(* Logix 5000 project; controller cal1615 1756-L62 rev 16.20; software revision 16.05; part 31 of 78 *)
(* tags used below, declared in another part *)
   AFI : BOOL;   // Always False Bit
   FAULT : BOOL;   // Fault AFI
   p01_param_fan_zero_speed : REAL;
   p01_param_open_oven_exh_sp : REAL;
   p01_param_open_oven_temp : REAL;
   p01_recipe_active : recipe;   // Active Recipe
   p01r09_open_oven : BOOL;
   p01r09_pb_global_reset : BOOL;   // System Modes PB: Global Fault Reset
   p02_dint_from_hmi : hmi_dint;
   p11r02_shutdown_temp : BOOL;   // Zone 1 Misc Control Safe Shutdown Temperature
   p11r30 : routine;   // Zone 1 Temperature Control
   p11r30_request_heat : BOOL;   // Zone 1 Temperature Control Request Heat
   p12r02_shutdown_temp : BOOL;   // Zone 2 Misc Control Safe Shutdown Temperature
   p12r30 : routine;   // Zone 2 Temperature Control
   p12r30_pid_temp : PID;   // Zone 2 Temperature Control PID
   p12r30_request_heat : BOOL;   // Zone 2 Temperature Control Request Heat
   p13_ai_exhaust_rpm : REAL;   // Zone 3 Analog Input Exhaust Fan RPM
   p13_ai_tc01 : REAL;   // Zone 3 Analog Input Control Thermocouple 1
   p13_ai_tc02 : REAL;   // Zone 3 Analog Input Control Thermocouple 2
   p13_ao_cv : REAL;   // Zone 3 Analog Output Control Valve
   p13_ao_exhaust_selected_speed : REAL;   // Zone 3 Analog Output Exhaust Fan VFD Selected Speed
   p13_di_door_open : BOOL;   // Zone 3 Digital Input Access Door Open
   p13_di_exh : acs800_di_normal;   // Zone 3 Digital Inputs Exhaust Fan
   p13_di_exh_fan_mtr_ts : BOOL;   // Zone 3 Digital Input Exhaust Fan Motor Thermostat OK
   p13_di_exh_flow_ok : BOOL;   // Zone 3 Digital Input Exhaust Flow OK
   p13_di_filter_clean : BOOL;   // Zone 3 Digital Input Filter Dirty
   p13_di_recirc : acs800_di_normal;   // Zone 3 Digital Inputs Recirc Fan
   p13_di_tc01_bo : BOOL;   // Zone 3 Digital Input Control Thermocouple 1 Failure
   p13_di_tc02_bo : BOOL;   // Zone 3 Digital Input Control Thermocouple 2 Failure
   p13_dint_to_hmi : DINT[16];   // Zone 3 Temperature Control VFDs On
   p13_do_exh : acs800_do_normal;   // Zone 3 Digital Output Exhaust Fan
   p13_param_pid2_ff : REAL;   // Zone 3 Parameter Auto PID Bias
   p13_param_pid2_kd : REAL;   // Zone 3 Parameter Auto PID Derivative Gain
   p13_param_pid2_ki : REAL;   // Zone 3 Parameter Auto PID Integral Gain
   p13_param_pid2_kp : REAL;   // Zone 3 Parameter Auto PID Proportional Gain
   p13_param_tc01_dev : REAL;   // Zone 3 Parameter Oven Temperature Deviation from Setpoint
   p13r01 : routine;   // Zone 3 Main
   p13r02_shutdown_temp : BOOL;   // Zone 3 Misc Control Safe Shutdown Temperature
   p13r16_pid_temp_cv : DINT;   // Zone 3 Temperature Control Control Valve
   p13r20_state : DINT;   // Zone 3 Temperature Control State
   p13r30 : routine;   // Zone 3 Temperature Control
   p13r30_cv_man_sp : REAL;   // Zone 3 Temperature Control Manual Heat Control Valve Setpoint
   p13r30_pb_auto : BOOL;   // Zone 3 Temperature Control PB: Zone Control Auto
   p13r30_pb_manual : BOOL;   // Zone 3 Temperature Control PB: Zone Control Manual
   p13r30_pb_zone_off : BOOL;   // Zone 3 Temperature Control PB: Stop Zone Heat Control
   p13r30_pb_zone_on : BOOL;   // Zone 3 Temperature Control PB: Start Zone Heat Control
   p13r30_permissive_run : BOOL;   // Zone 3 Temperature Control Run Permissive
   p13r30_pid_temp_pv : REAL;   // Zone 3 Temperature Control PID Process Value
   p13r30_pid_temp_sp : REAL;   // Zone 3 Temperature Control PID Temperature Control Setpoint
   p13r30_pid_temp_sp_error : REAL;   // Zone 3 Temperature Control Setpoint/Process Variable Error (ABS)
   p13r30_pid_temp_sp_last : REAL;   // Zone 3 Temperature Control Setpoint Last Scan
   p13r30_request_cool : BOOL;   // Zone 3 Temperature Control Request Cooling
   p13r30_request_deviation_warning : BOOL;   // Zone 3 Temperature Control Request Setpoint Deviation Warning
   p13r30_request_manual : BOOL;   // Zone 3 Temperature Control Request Manual Control
   p13r30_request_PID_shot : BOOL;
   p13r30_temp_deviation_setpoint : DINT;
   p13r30_temp_pid_ctrl : PID;   // Zone 3 Temperature Control PID
   p13r30_timer_fault : TIMER[16];   // Zone 3 Temperature Control Fault Delay
   p13r30_timer_warning : TIMER[12];   // Zone 3 Temperature Control Warning Delay
   p13r30_vfds_ready : BOOL;   // Zone 3 Temperature Control VFDs On
   p13r31 : routine;   // Zone 3 Exhaust VFD
   p13r31_pb_start : BOOL;   // Zone 3 Exhaust VFD PB: Start
   p13r31_pb_stop : BOOL;   // Zone 3 Exhaust VFD PB: Stop
   p13r31_request_auto_run : BOOL;   // Zone 3 Exhaust Fan Run Request
   p13r31_run_permissive : BOOL;   // Zone 3 Exhaust VFD Run Permissive
   p13r31_timer_fault : TIMER[5];   // Zone 3 Exhaust VFD Fault Timer
   p13r31_timer_warning : TIMER[5];   // Zone 3 Exhaust VFD Waringing Timer
   p13r31_vfd_stopped : BOOL;   // Zone 3 Exhaust VFD VFD Stopped
   p23r02 : routine;   // Impreg Misc Control
(* P13_Zone_3, continued *)

ROUTINE R30_Temperature_Control   (* ladder *)
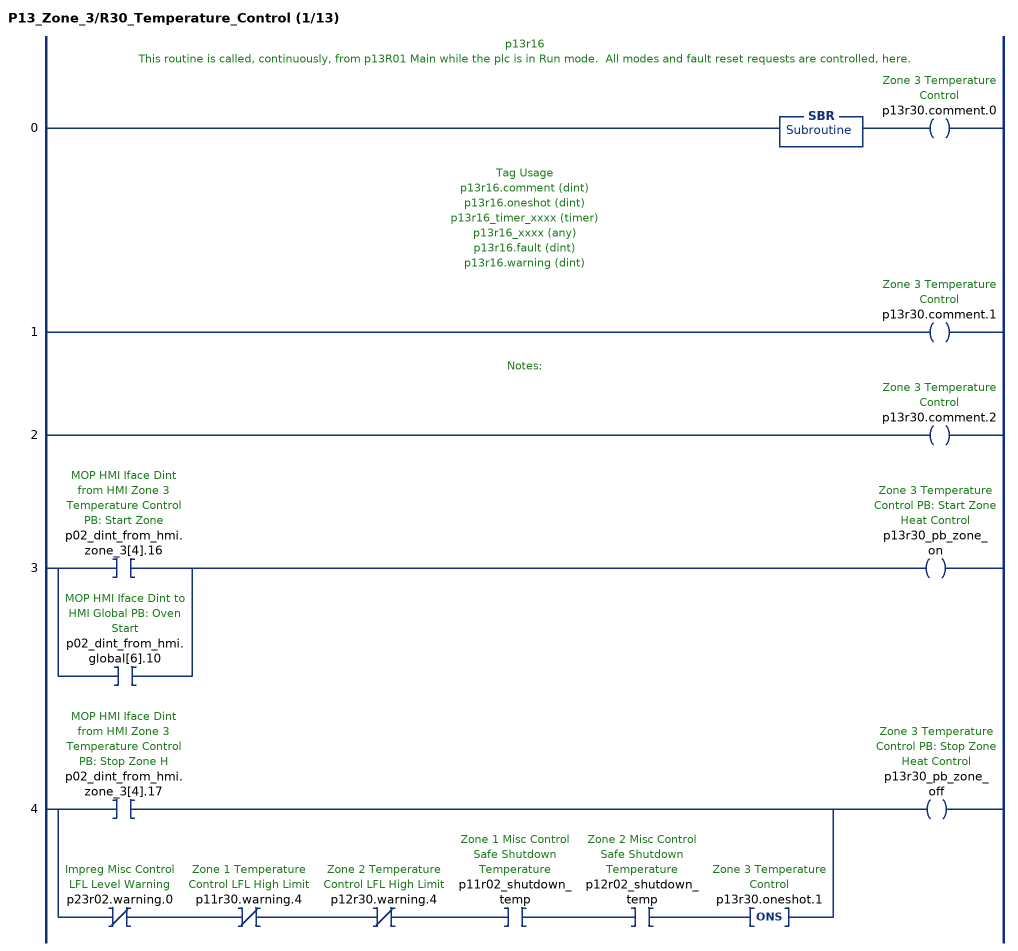
   // p13r16
   // This routine is called, continuously, from p13R01 Main while the plc is in Run mode.  All modes and fault reset requests are controlled, here.
   0: SBR()OTE(p13r30.comment.0);
   // Tag Usage
   // p13r16.comment (dint)
   // p13r16.oneshot (dint)
   // p13r16_timer_xxxx (timer)
   // p13r16_xxxx (any)
   // p13r16.fault (dint)
   // p13r16.warning (dint)
   1: OTE(p13r30.comment.1);
   // Notes:
   2: OTE(p13r30.comment.2);
   3: [XIC(p02_dint_from_hmi.zone_3[4].16) ,XIC(p02_dint_from_hmi.global[6].10) ]OTE(p13r30_pb_zone_on);
   4: [XIC(p02_dint_from_hmi.zone_3[4].17) ,XIO(p23r02.warning.0) XIO(p11r30.warning.4) XIO(p12r30.warning.4) XIC(p11r02_shutdown_temp) XIC(p12r02_shutdown_temp) ONS(p13r30.oneshot.1) ]OTE(p13r30_pb_zone_off);
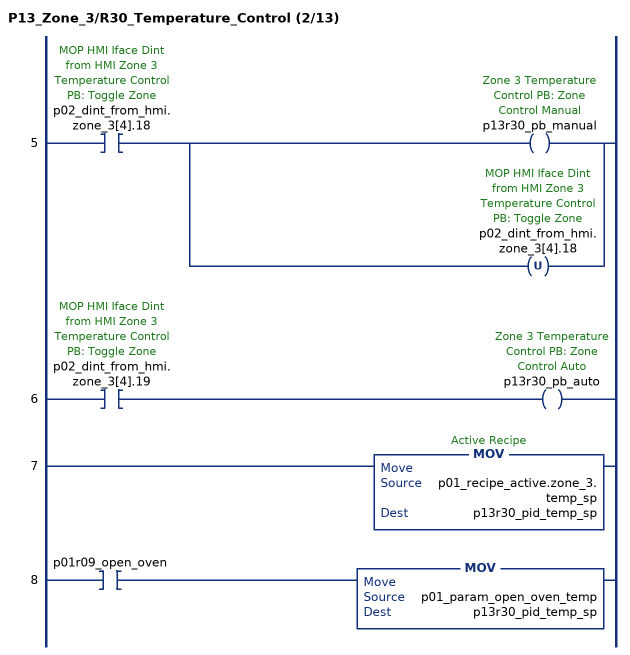
   5: XIC(p02_dint_from_hmi.zone_3[4].18)[OTE(p13r30_pb_manual) ,OTU(p02_dint_from_hmi.zone_3[4].18) ];
   6: XIC(p02_dint_from_hmi.zone_3[4].19)OTE(p13r30_pb_auto);
   7: MOV(p01_recipe_active.zone_3.temp_sp,p13r30_pid_temp_sp);
   8: XIC(p01r09_open_oven)MOV(p01_param_open_oven_temp,p13r30_pid_temp_sp);
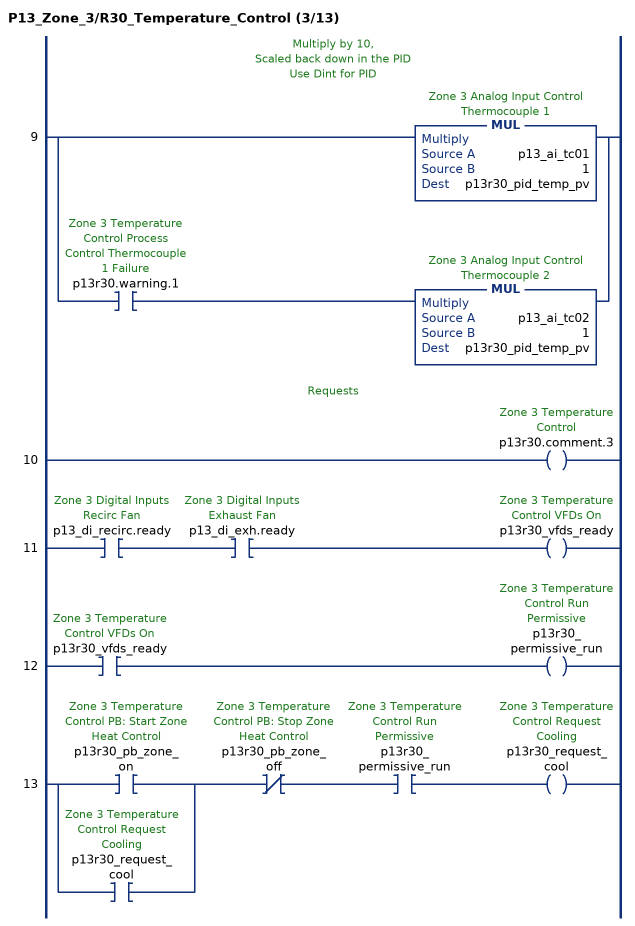
   // Multiply by 10,
   // Scaled back down in the PID
   // Use Dint for PID
   9: [MUL(p13_ai_tc01,1,p13r30_pid_temp_pv) ,XIC(p13r30.warning.1) MUL(p13_ai_tc02,1,p13r30_pid_temp_pv) ];
   // Requests
   10: OTE(p13r30.comment.3);
   11: XIC(p13_di_recirc.ready)XIC(p13_di_exh.ready)OTE(p13r30_vfds_ready);
   12: XIC(p13r30_vfds_ready)OTE(p13r30_permissive_run);
   13: [XIC(p13r30_pb_zone_on) ,XIC(p13r30_request_cool) ]XIO(p13r30_pb_zone_off)XIC(p13r30_permissive_run)OTE(p13r30_request_cool);
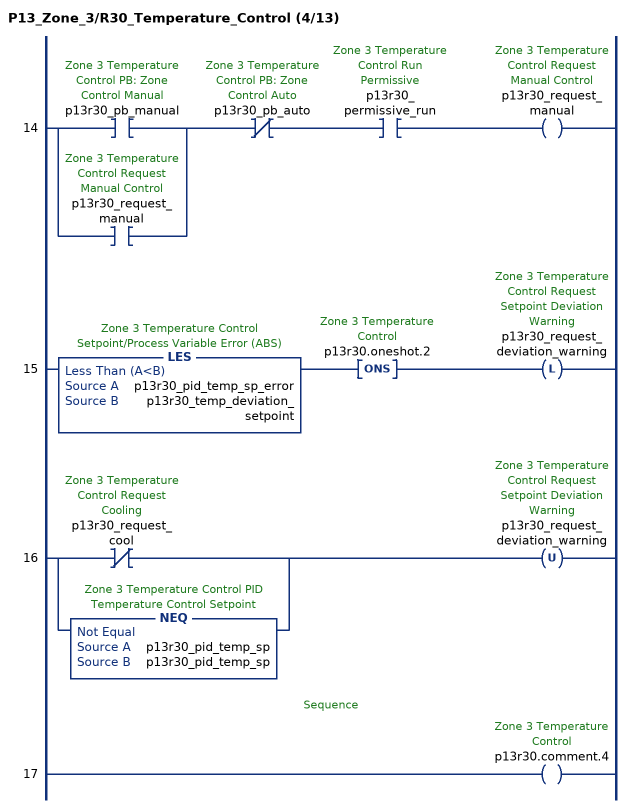
   14: [XIC(p13r30_pb_manual) ,XIC(p13r30_request_manual) ]XIO(p13r30_pb_auto)XIC(p13r30_permissive_run)OTE(p13r30_request_manual);
   15: LES(p13r30_pid_temp_sp_error,p13r30_temp_deviation_setpoint)ONS(p13r30.oneshot.2)OTL(p13r30_request_deviation_warning);
   16: [XIO(p13r30_request_cool) ,NEQ(p13r30_pid_temp_sp,p13r30_pid_temp_sp) ]OTU(p13r30_request_deviation_warning);
   // Sequence
   17: OTE(p13r30.comment.4);
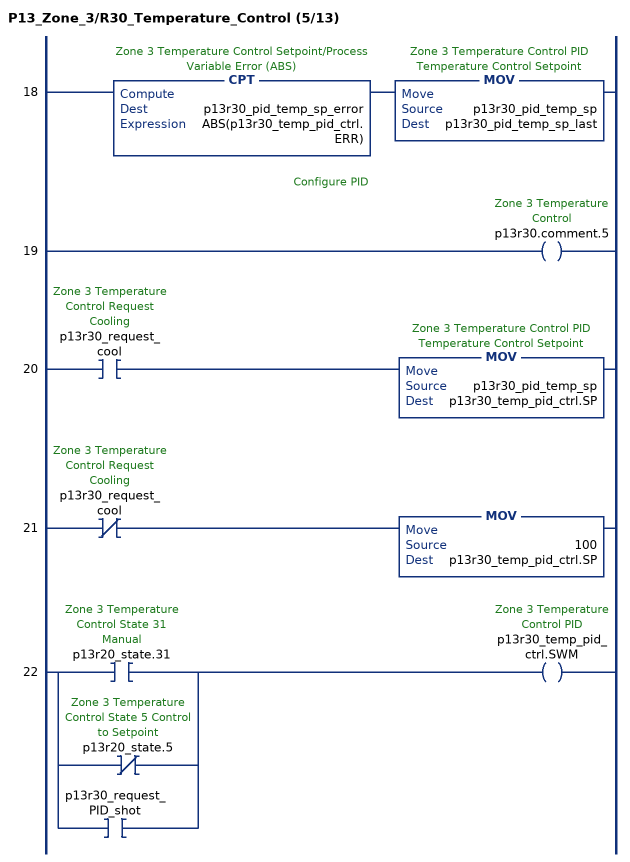
   18: CPT(p13r30_pid_temp_sp_error,ABS(p13r30_temp_pid_ctrl.ERR))MOV(p13r30_pid_temp_sp,p13r30_pid_temp_sp_last);
   // Configure PID
   19: OTE(p13r30.comment.5);
   20: XIC(p13r30_request_cool)MOV(p13r30_pid_temp_sp,p13r30_temp_pid_ctrl.SP);
   21: XIO(p13r30_request_cool)MOV(100,p13r30_temp_pid_ctrl.SP);
   22: [XIC(p13r20_state.31) ,XIO(p13r20_state.5) ,XIC(p13r30_request_PID_shot) ]OTE(p13r30_temp_pid_ctrl.SWM);
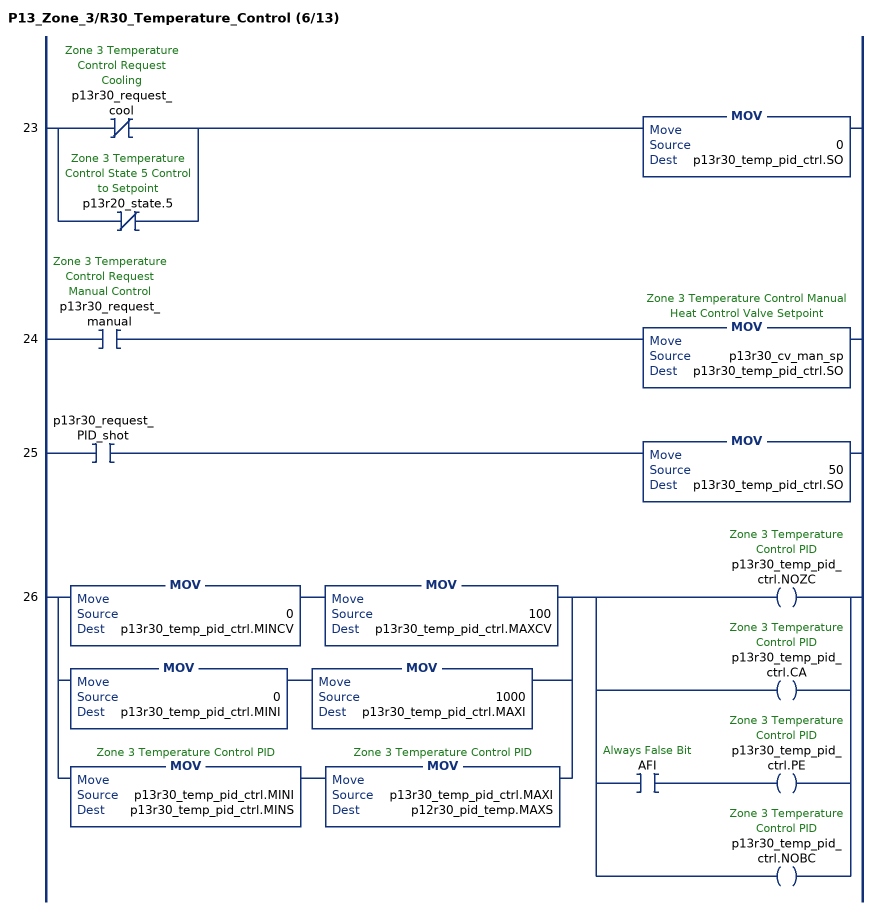
   23: [XIO(p13r30_request_cool) ,XIO(p13r20_state.5) ]MOV(0,p13r30_temp_pid_ctrl.SO);
   24: XIC(p13r30_request_manual)MOV(p13r30_cv_man_sp,p13r30_temp_pid_ctrl.SO);
   25: XIC(p13r30_request_PID_shot)MOV(50,p13r30_temp_pid_ctrl.SO);
   26: [MOV(0,p13r30_temp_pid_ctrl.MINCV) MOV(100,p13r30_temp_pid_ctrl.MAXCV) ,MOV(0,p13r30_temp_pid_ctrl.MINI) MOV(1000,p13r30_temp_pid_ctrl.MAXI) ,MOV(p13r30_temp_pid_ctrl.MINI,p13r30_temp_pid_ctrl.MINS) MOV(p13r30_temp_pid_ctrl.MAXI,p12r30_pid_temp.MAXS) ][OTE(p13r30_temp_pid_ctrl.NOZC) ,OTE(p13r30_temp_pid_ctrl.CA) ,XIC(AFI) OTE(p13r30_temp_pid_ctrl.PE) ,OTE(p13r30_temp_pid_ctrl.NOBC) ];
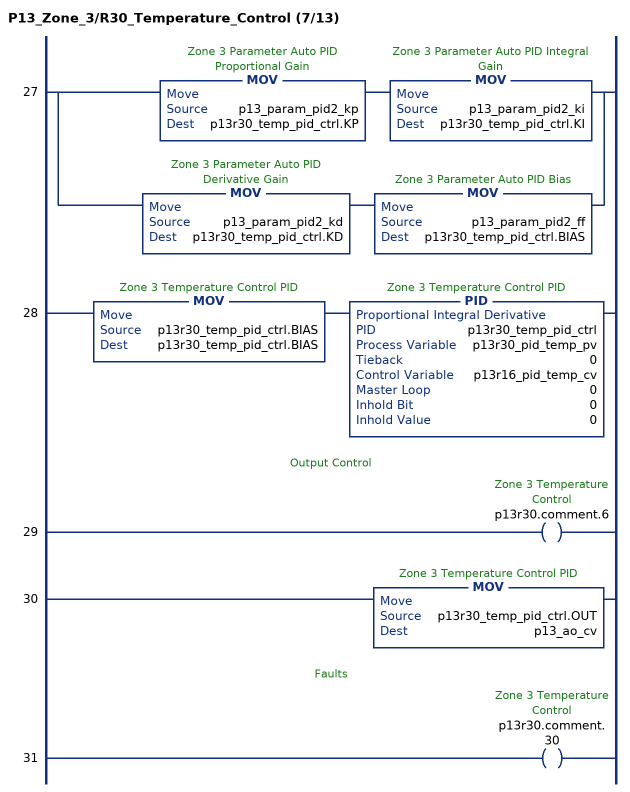
   27: [MOV(p13_param_pid2_kp,p13r30_temp_pid_ctrl.KP) MOV(p13_param_pid2_ki,p13r30_temp_pid_ctrl.KI) ,MOV(p13_param_pid2_kd,p13r30_temp_pid_ctrl.KD) MOV(p13_param_pid2_ff,p13r30_temp_pid_ctrl.BIAS) ];
   28: MOV(p13r30_temp_pid_ctrl.BIAS,p13r30_temp_pid_ctrl.BIAS)PID(p13r30_temp_pid_ctrl,p13r30_pid_temp_pv,0,p13r16_pid_temp_cv,0,0,0);
   // Output Control
   29: OTE(p13r30.comment.6);
   30: MOV(p13r30_temp_pid_ctrl.OUT,p13_ao_cv);
   // Faults
   31: OTE(p13r30.comment.30);
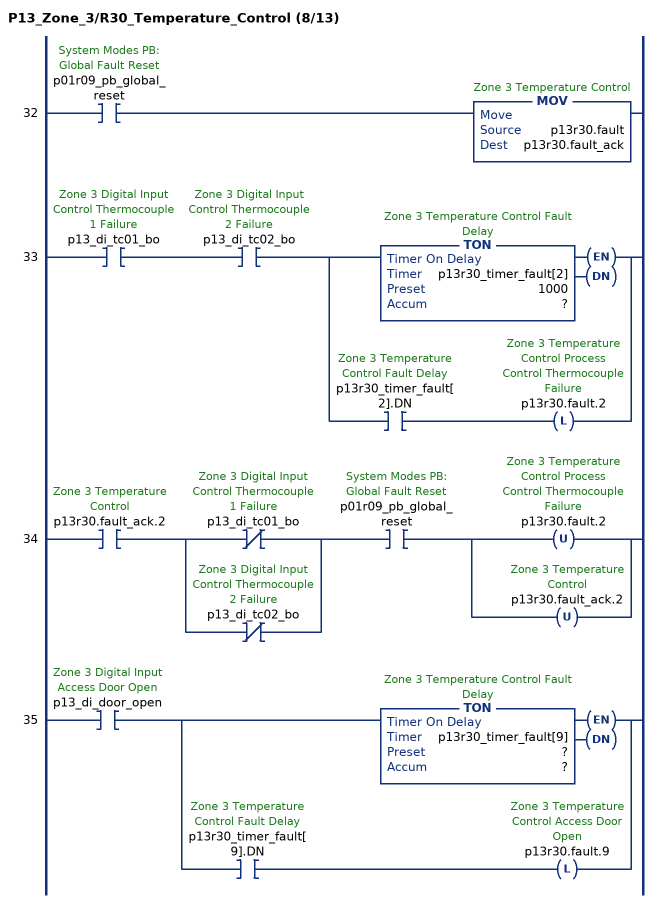
   32: XIC(p01r09_pb_global_reset)MOV(p13r30.fault,p13r30.fault_ack);
   33: XIC(p13_di_tc01_bo)XIC(p13_di_tc02_bo)[TON(p13r30_timer_fault[2],?,?) ,XIC(p13r30_timer_fault[2].DN) OTL(p13r30.fault.2) ];
   34: XIC(p13r30.fault_ack.2)[XIO(p13_di_tc01_bo) ,XIO(p13_di_tc02_bo) ]XIC(p01r09_pb_global_reset)[OTU(p13r30.fault.2) ,OTU(p13r30.fault_ack.2) ];
   35: XIC(p13_di_door_open)[TON(p13r30_timer_fault[9],?,?) ,XIC(p13r30_timer_fault[9].DN) OTL(p13r30.fault.9) ];
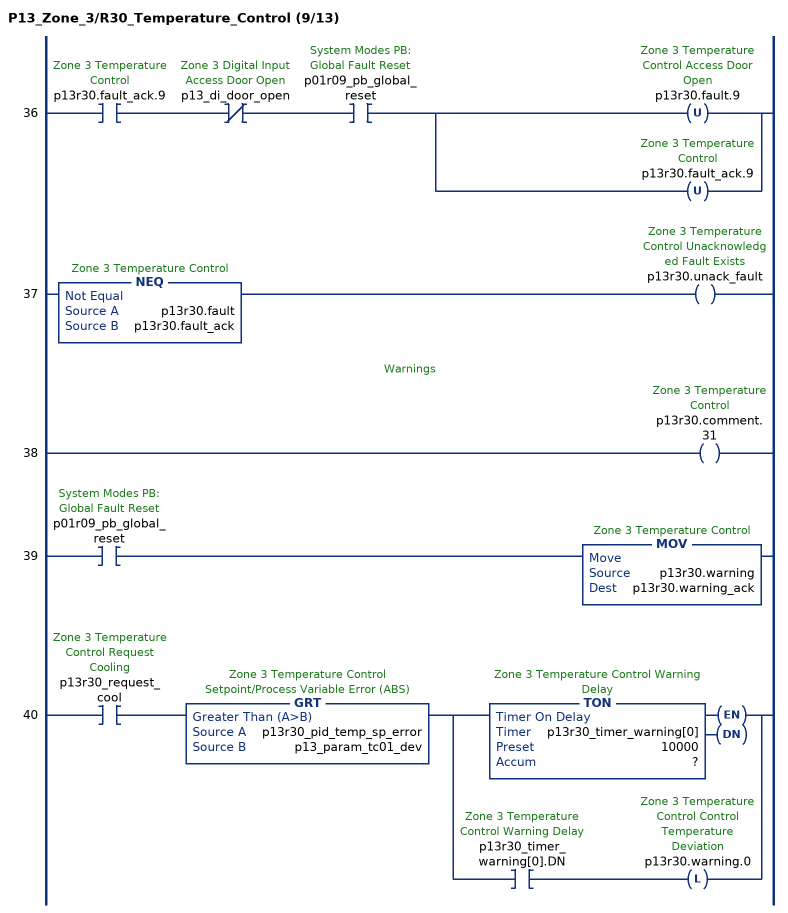
   36: XIC(p13r30.fault_ack.9)XIO(p13_di_door_open)XIC(p01r09_pb_global_reset)[OTU(p13r30.fault.9) ,OTU(p13r30.fault_ack.9) ];
   37: NEQ(p13r30.fault,p13r30.fault_ack)OTE(p13r30.unack_fault);
   // Warnings
   38: OTE(p13r30.comment.31);
   39: XIC(p01r09_pb_global_reset)MOV(p13r30.warning,p13r30.warning_ack);
   40: XIC(p13r30_request_cool)GRT(p13r30_pid_temp_sp_error,p13_param_tc01_dev)[TON(p13r30_timer_warning[0],?,?) ,XIC(p13r30_timer_warning[0].DN) OTL(p13r30.warning.0) ];
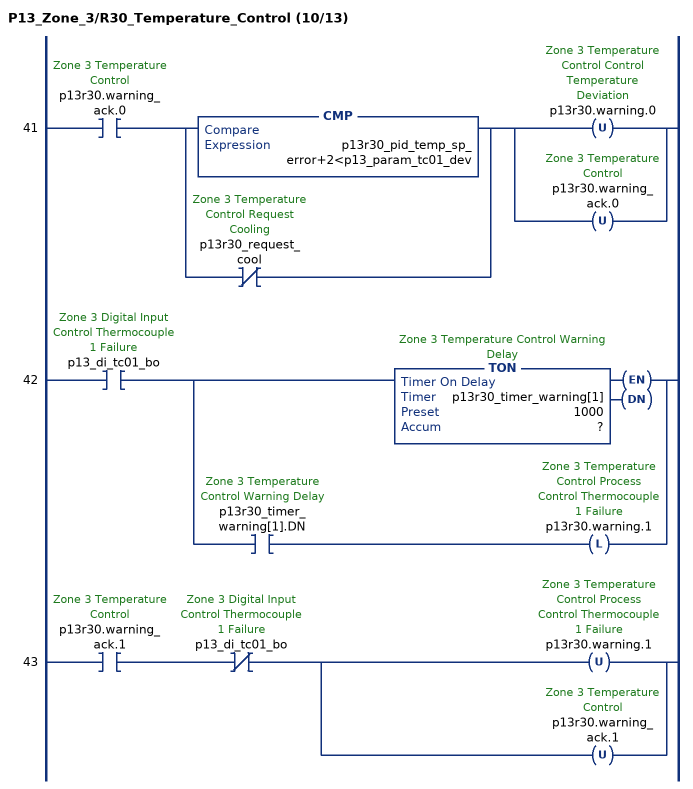
   41: XIC(p13r30.warning_ack.0)[CMP(p13r30_pid_temp_sp_error+2<p13_param_tc01_dev) ,XIO(p13r30_request_cool) ][OTU(p13r30.warning.0) ,OTU(p13r30.warning_ack.0) ];
   42: XIC(p13_di_tc01_bo)[TON(p13r30_timer_warning[1],?,?) ,XIC(p13r30_timer_warning[1].DN) OTL(p13r30.warning.1) ];
   43: XIC(p13r30.warning_ack.1)XIO(p13_di_tc01_bo)[OTU(p13r30.warning.1) ,OTU(p13r30.warning_ack.1) ];
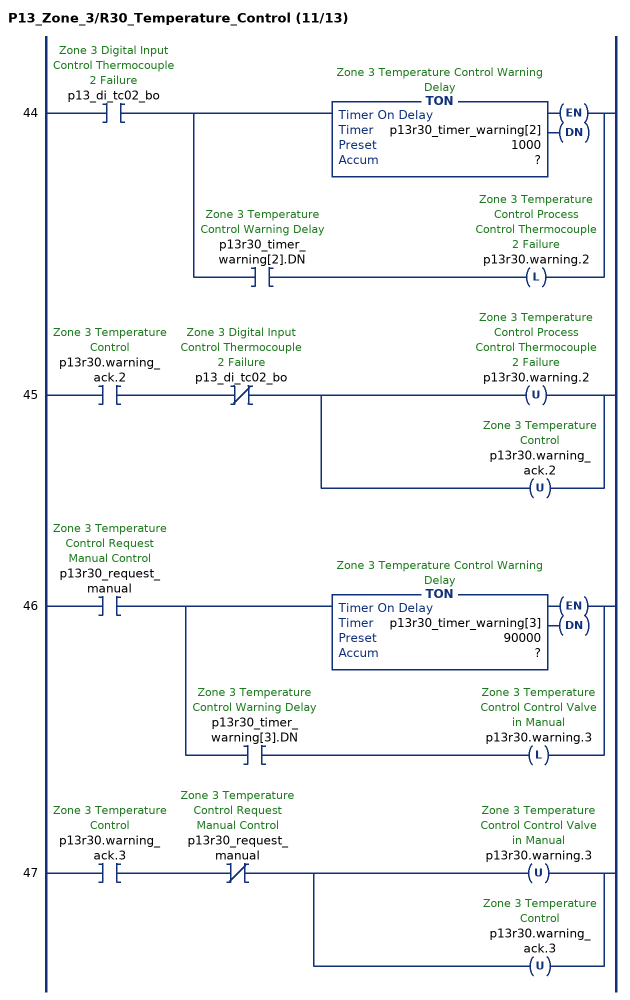
   44: XIC(p13_di_tc02_bo)[TON(p13r30_timer_warning[2],?,?) ,XIC(p13r30_timer_warning[2].DN) OTL(p13r30.warning.2) ];
   45: XIC(p13r30.warning_ack.2)XIO(p13_di_tc02_bo)[OTU(p13r30.warning.2) ,OTU(p13r30.warning_ack.2) ];
   46: XIC(p13r30_request_manual)[TON(p13r30_timer_warning[3],?,?) ,XIC(p13r30_timer_warning[3].DN) OTL(p13r30.warning.3) ];
   47: XIC(p13r30.warning_ack.3)XIO(p13r30_request_manual)[OTU(p13r30.warning.3) ,OTU(p13r30.warning_ack.3) ];
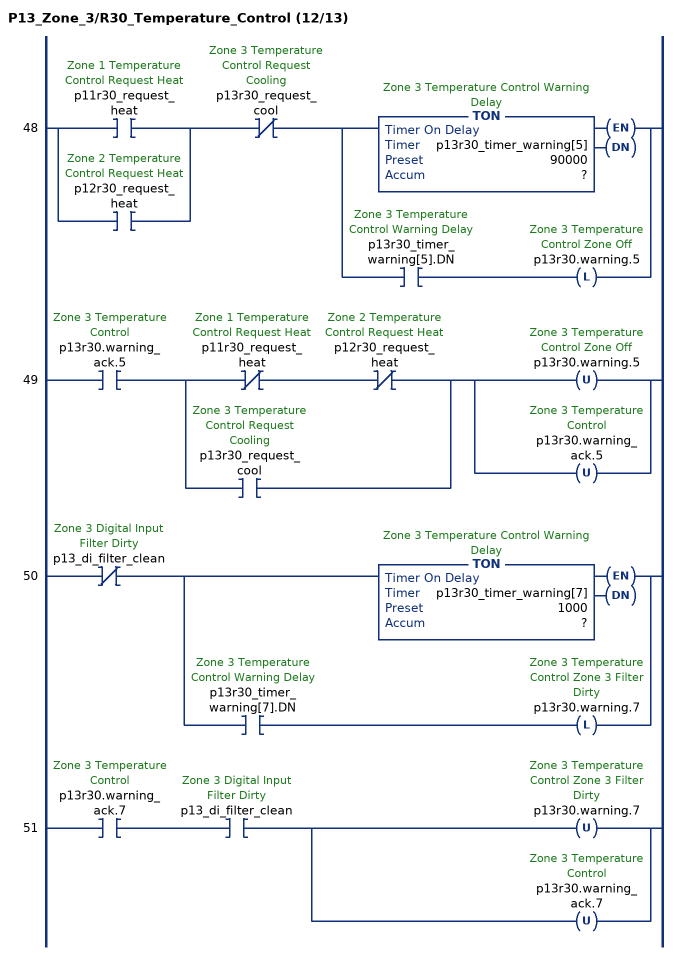
   48: [XIC(p11r30_request_heat) ,XIC(p12r30_request_heat) ]XIO(p13r30_request_cool)[TON(p13r30_timer_warning[5],?,?) ,XIC(p13r30_timer_warning[5].DN) OTL(p13r30.warning.5) ];
   49: XIC(p13r30.warning_ack.5)[XIO(p11r30_request_heat) XIO(p12r30_request_heat) ,XIC(p13r30_request_cool) ][OTU(p13r30.warning.5) ,OTU(p13r30.warning_ack.5) ];
   50: XIO(p13_di_filter_clean)[TON(p13r30_timer_warning[7],?,?) ,XIC(p13r30_timer_warning[7].DN) OTL(p13r30.warning.7) ];
   51: XIC(p13r30.warning_ack.7)XIC(p13_di_filter_clean)[OTU(p13r30.warning.7) ,OTU(p13r30.warning_ack.7) ];
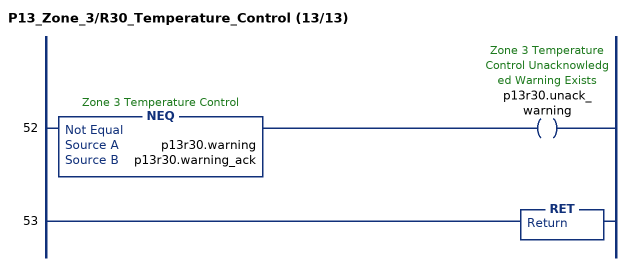
   52: NEQ(p13r30.warning,p13r30.warning_ack)OTE(p13r30.unack_warning);
   53: RET();
END_ROUTINE

ROUTINE R31_Exhaust_VFD   (* ladder *)
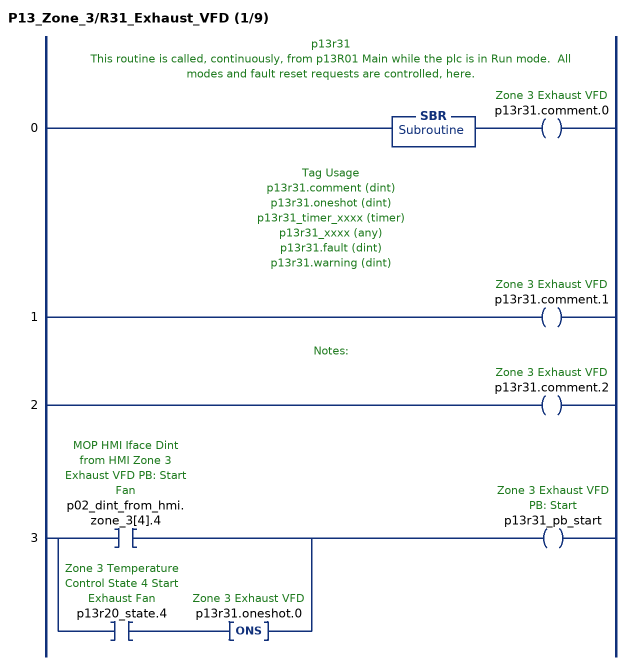
   // p13r31
   // This routine is called, continuously, from p13R01 Main while the plc is in Run mode.  All modes and fault reset requests are controlled, here.
   0: SBR()OTE(p13r31.comment.0);
   // Tag Usage
   // p13r31.comment (dint)
   // p13r31.oneshot (dint)
   // p13r31_timer_xxxx (timer)
   // p13r31_xxxx (any)
   // p13r31.fault (dint)
   // p13r31.warning (dint)
   1: OTE(p13r31.comment.1);
   // Notes:
   2: OTE(p13r31.comment.2);
   3: [XIC(p02_dint_from_hmi.zone_3[4].4) ,XIC(p13r20_state.4) ONS(p13r31.oneshot.0) ]OTE(p13r31_pb_start);
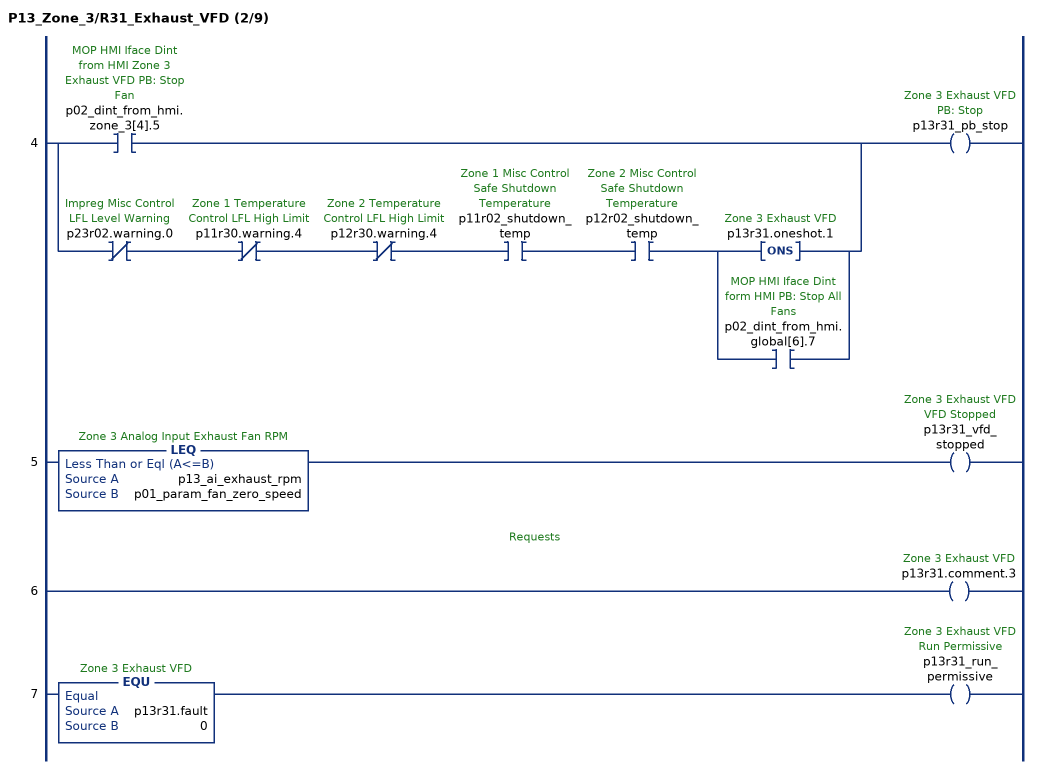
   4: [XIC(p02_dint_from_hmi.zone_3[4].5) ,XIO(p23r02.warning.0) XIO(p11r30.warning.4) XIO(p12r30.warning.4) XIC(p11r02_shutdown_temp) XIC(p12r02_shutdown_temp) [ONS(p13r31.oneshot.1) ,XIC(p02_dint_from_hmi.global[6].7) ] ]OTE(p13r31_pb_stop);
   5: LEQ(p13_ai_exhaust_rpm,p01_param_fan_zero_speed)OTE(p13r31_vfd_stopped);
   // Requests
   6: OTE(p13r31.comment.3);
   7: EQU(p13r31.fault,0)OTE(p13r31_run_permissive);
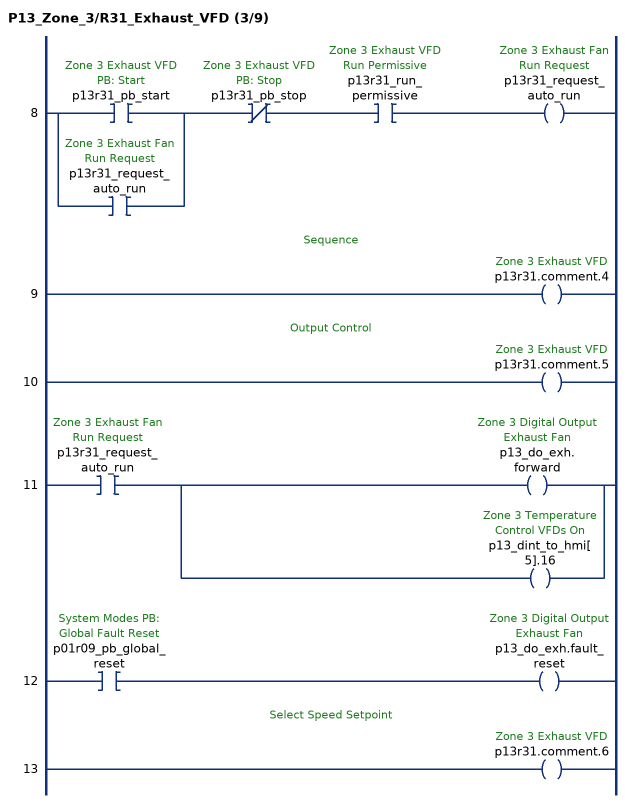
   8: [XIC(p13r31_pb_start) ,XIC(p13r31_request_auto_run) ]XIO(p13r31_pb_stop)XIC(p13r31_run_permissive)OTE(p13r31_request_auto_run);
   // Sequence
   9: OTE(p13r31.comment.4);
   // Output Control
   10: OTE(p13r31.comment.5);
   11: XIC(p13r31_request_auto_run)[OTE(p13_do_exh.forward) ,OTE(p13_dint_to_hmi[5].16) ];
   12: XIC(p01r09_pb_global_reset)OTE(p13_do_exh.fault_reset);
   // Select Speed Setpoint
   13: OTE(p13r31.comment.6);
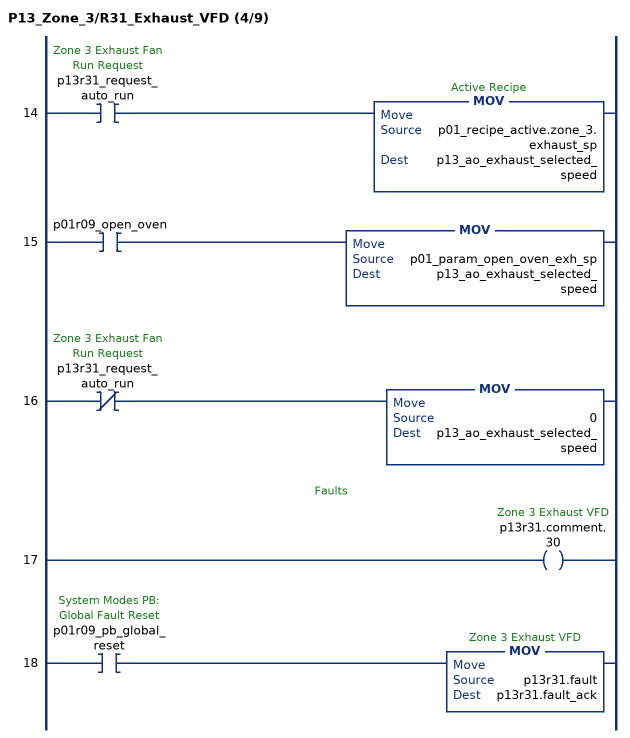
   14: XIC(p13r31_request_auto_run)MOV(p01_recipe_active.zone_3.exhaust_sp,p13_ao_exhaust_selected_speed);
   15: XIC(p01r09_open_oven)MOV(p01_param_open_oven_exh_sp,p13_ao_exhaust_selected_speed);
   16: XIO(p13r31_request_auto_run)MOV(0,p13_ao_exhaust_selected_speed);
   // Faults
   17: OTE(p13r31.comment.30);
   18: XIC(p01r09_pb_global_reset)MOV(p13r31.fault,p13r31.fault_ack);
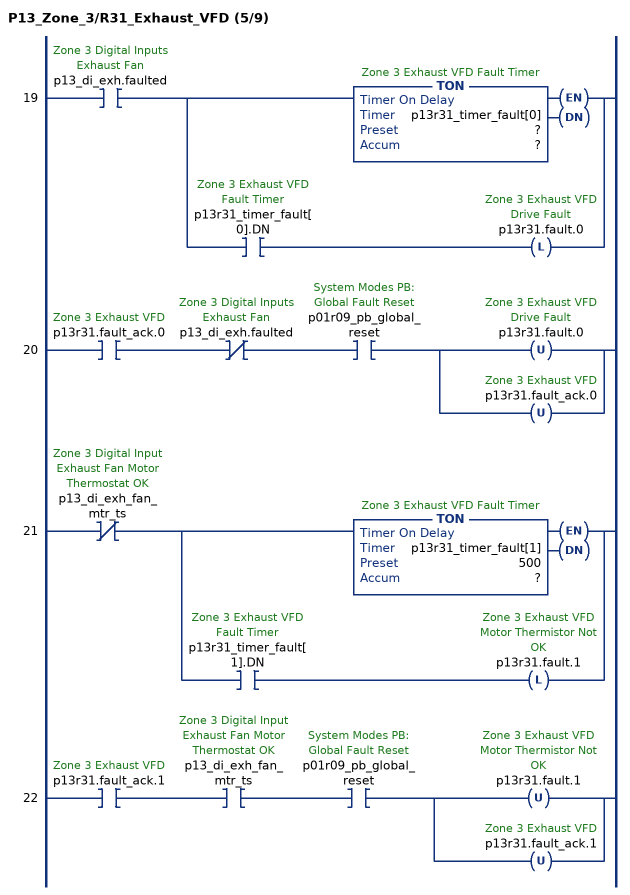
   19: XIC(p13_di_exh.faulted)[TON(p13r31_timer_fault[0],?,?) ,XIC(p13r31_timer_fault[0].DN) OTL(p13r31.fault.0) ];
   20: XIC(p13r31.fault_ack.0)XIO(p13_di_exh.faulted)XIC(p01r09_pb_global_reset)[OTU(p13r31.fault.0) ,OTU(p13r31.fault_ack.0) ];
   21: XIO(p13_di_exh_fan_mtr_ts)[TON(p13r31_timer_fault[1],?,?) ,XIC(p13r31_timer_fault[1].DN) OTL(p13r31.fault.1) ];
   22: XIC(p13r31.fault_ack.1)XIC(p13_di_exh_fan_mtr_ts)XIC(p01r09_pb_global_reset)[OTU(p13r31.fault.1) ,OTU(p13r31.fault_ack.1) ];
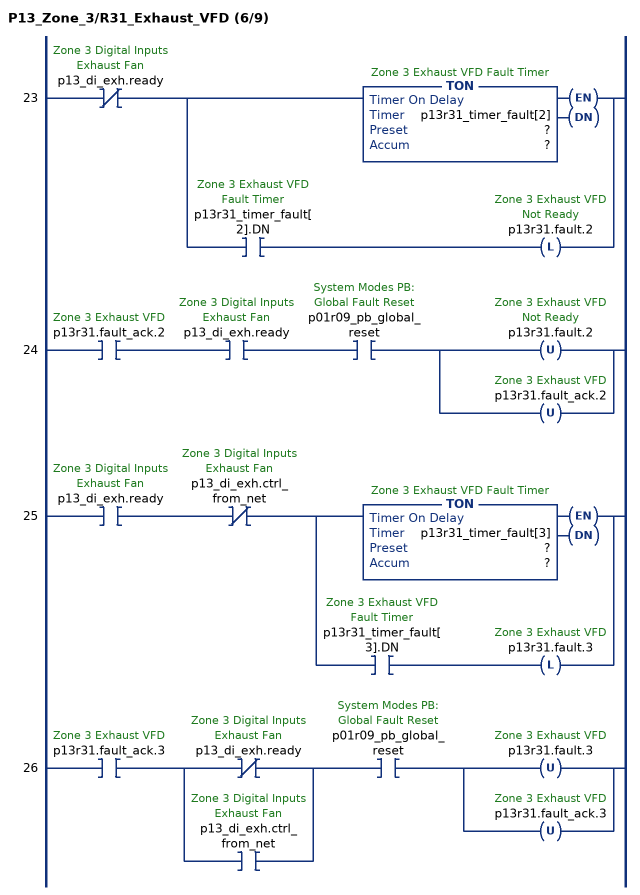
   23: XIO(p13_di_exh.ready)[TON(p13r31_timer_fault[2],?,?) ,XIC(p13r31_timer_fault[2].DN) OTL(p13r31.fault.2) ];
   24: XIC(p13r31.fault_ack.2)XIC(p13_di_exh.ready)XIC(p01r09_pb_global_reset)[OTU(p13r31.fault.2) ,OTU(p13r31.fault_ack.2) ];
   25: XIC(p13_di_exh.ready)XIO(p13_di_exh.ctrl_from_net)[TON(p13r31_timer_fault[3],?,?) ,XIC(p13r31_timer_fault[3].DN) OTL(p13r31.fault.3) ];
   26: XIC(p13r31.fault_ack.3)[XIO(p13_di_exh.ready) ,XIC(p13_di_exh.ctrl_from_net) ]XIC(p01r09_pb_global_reset)[OTU(p13r31.fault.3) ,OTU(p13r31.fault_ack.3) ];
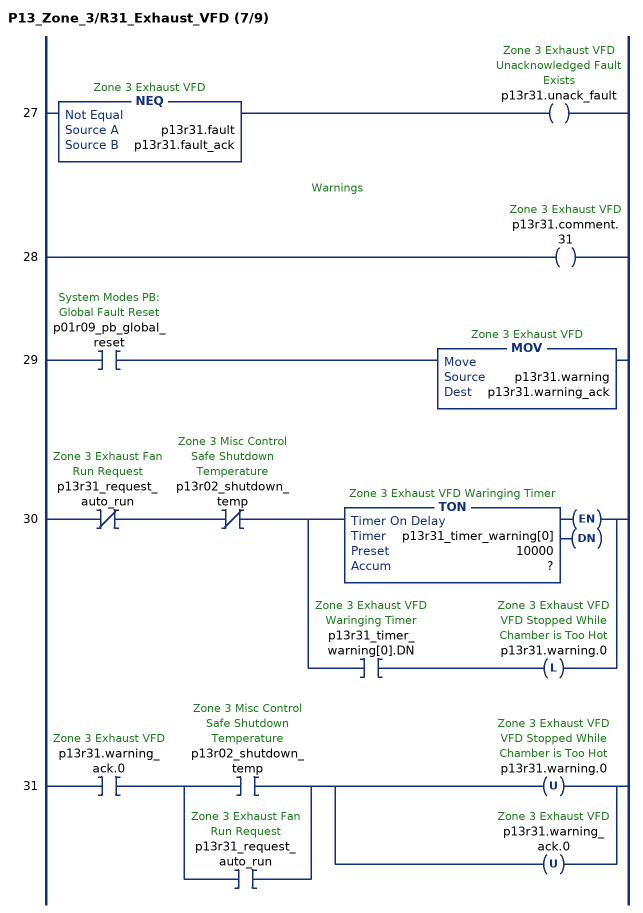
   27: NEQ(p13r31.fault,p13r31.fault_ack)OTE(p13r31.unack_fault);
   // Warnings
   28: OTE(p13r31.comment.31);
   29: XIC(p01r09_pb_global_reset)MOV(p13r31.warning,p13r31.warning_ack);
   30: XIO(p13r31_request_auto_run)XIO(p13r02_shutdown_temp)[TON(p13r31_timer_warning[0],?,?) ,XIC(p13r31_timer_warning[0].DN) OTL(p13r31.warning.0) ];
   31: XIC(p13r31.warning_ack.0)[XIC(p13r02_shutdown_temp) ,XIC(p13r31_request_auto_run) ][OTU(p13r31.warning.0) ,OTU(p13r31.warning_ack.0) ];
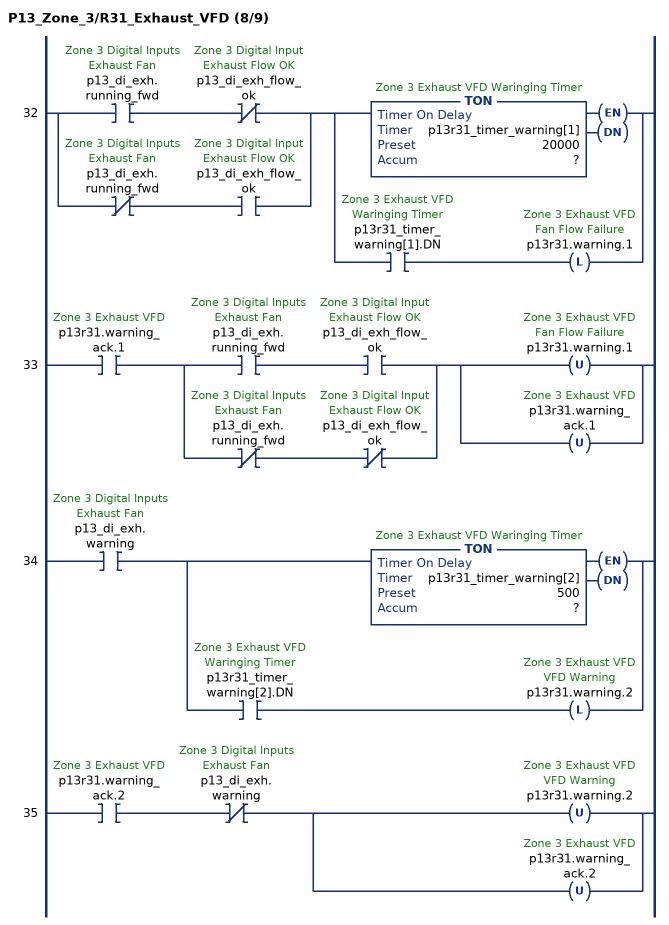
   32: [XIC(p13_di_exh.running_fwd) XIO(p13_di_exh_flow_ok) ,XIO(p13_di_exh.running_fwd) XIC(p13_di_exh_flow_ok) ][TON(p13r31_timer_warning[1],?,?) ,XIC(p13r31_timer_warning[1].DN) OTL(p13r31.warning.1) ];
   33: XIC(p13r31.warning_ack.1)[XIC(p13_di_exh.running_fwd) XIC(p13_di_exh_flow_ok) ,XIO(p13_di_exh.running_fwd) XIO(p13_di_exh_flow_ok) ][OTU(p13r31.warning.1) ,OTU(p13r31.warning_ack.1) ];
   34: XIC(p13_di_exh.warning)[TON(p13r31_timer_warning[2],?,?) ,XIC(p13r31_timer_warning[2].DN) OTL(p13r31.warning.2) ];
   35: XIC(p13r31.warning_ack.2)XIO(p13_di_exh.warning)[OTU(p13r31.warning.2) ,OTU(p13r31.warning_ack.2) ];
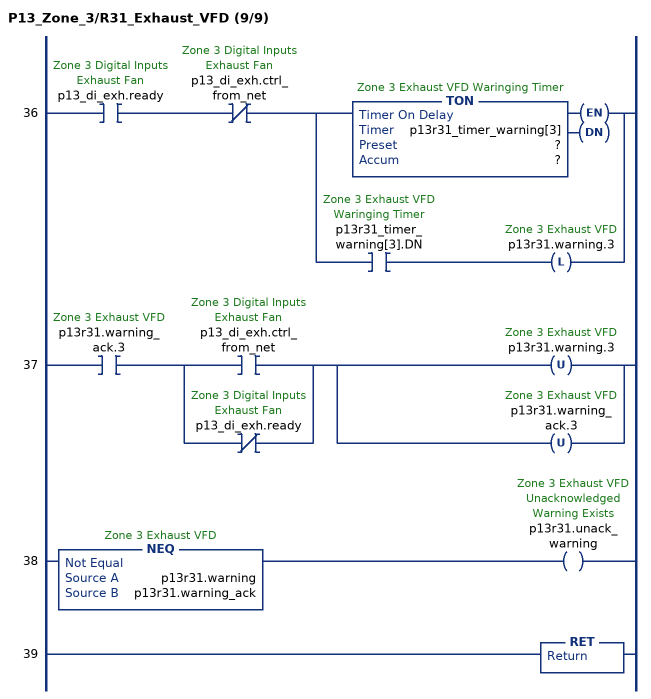
   36: XIC(p13_di_exh.ready)XIO(p13_di_exh.ctrl_from_net)[TON(p13r31_timer_warning[3],?,?) ,XIC(p13r31_timer_warning[3].DN) OTL(p13r31.warning.3) ];
   37: XIC(p13r31.warning_ack.3)[XIC(p13_di_exh.ctrl_from_net) ,XIO(p13_di_exh.ready) ][OTU(p13r31.warning.3) ,OTU(p13r31.warning_ack.3) ];
   38: NEQ(p13r31.warning,p13r31.warning_ack)OTE(p13r31.unack_warning);
   39: RET();
END_ROUTINE
